// Mitsubishi GX Works2 project: Termin3_Drugi_zadatak   PLC: FX3S

// task Task_01 (event TRUE, interval 0, priority 31): POU_01

PROGRAM POU_01
VAR
  induktivni_senzor : BOOL;
  TON_1 : TON;
  vreme_tajmera1 : TIME;
  Tizl1 : BOOL;
  TON_2 : TON;
  vreme_tajmera2 : TIME;
  Tizl2 : BOOL;
  Motor : BOOL;
END_VAR
(* structured ladder/FBD written out as ST: instructions are called as NAME(EN, inputs, outputs); _pN, _eN, _tN stand for wires *)
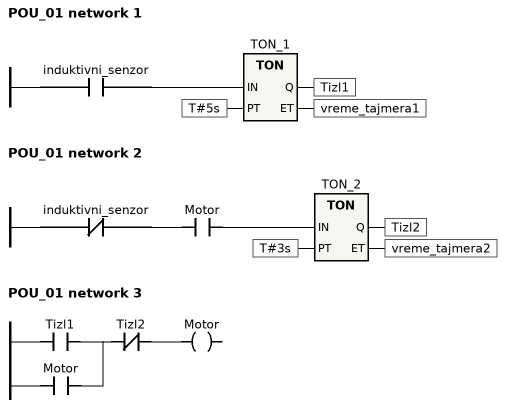
(* network 1 *)
TON_1(IN := induktivni_senzor, PT := T#5s, Q => Tizl1, ET => vreme_tajmera1);
(* network 2 *)
TON_2(IN := NOT induktivni_senzor AND Motor, PT := T#3s, Q => Tizl2, ET => vreme_tajmera2);
(* network 3 *)
Motor := (Tizl1 OR Motor) AND NOT Tizl2;
END_PROGRAM
